PROGRAM LateBlanking_Scan
VAR
	CS_CodeTcp_cold: CS_CodeTcp;
	Cold_step :UINT;
	scan_TON1 :Tc2_Standard.TON;
	Scan_TON :ARRAY[1..7] OF Tc2_Standard.TON;
	Scan_code_Z : R_TRIG;
	I:INT;
END_VAR

//扫码



Saoma();
P3User2_Par.Scan_IP:='192.168.10.26';
Scan_TON[1](PT:=T#1MS);
Scan_TON[2](PT:=T#1MS);
Scan_TON[3](PT:=T#1MS);
Scan_TON[4](PT:=T#100MS);

Scan_code_Z (CLK:=Cold_Scan_code, Q=>);

IF Scan_code_Z.Q AND  Cold_step=0 THEN
	 Cold_step:=10;
END_IF




CASE Cold_step OF
0:
	IF Scan_start AND NOT bCodeError AND NOT bCodeConError AND NOT P3User2_Par.Shield[4] THEN
	 Cold_step:=10;
	 Code_State:=0;
	ELSIF P3User2_Par.Shield[4] THEN
	 Cold_step:=70;
	END_IF
10:
	Scan_TON[1].IN:=FALSE;
	Scan_TON[2].IN:=FALSE;
	Scan_TON[3].IN:=FALSE;
	Cold_step:=20;
	
20:
	bScan_init:=TRUE;
	Scan_TON[1].IN:=TRUE;
	IF Scan_TON[1].Q THEN
		bScan_init:=FALSE;
		Scan_TON[1].IN:=FALSE;
		Cold_step:=30;
	END_IF

30:
	bTcpOpen:=TRUE;
	Scan_TON[2].IN:=TRUE;
	IF Scan_TON[2].Q THEN
		bTcpOpen:=FALSE;
		Scan_TON[2].IN:=FALSE;
		Cold_step:=40;
	END_IF

40:
	IF bTcpOpen_OK THEN
		Cold_step:=50;
	END_IF

50:
	bScan_start:=TRUE;
	Scan_TON[3].IN:=TRUE;
	IF Scan_TON[3].Q THEN
		bScan_start:=FALSE;
		Scan_TON[3].IN:=FALSE;
		Cold_step:=60;
	END_IF
60:
	Scan_TON[4].IN:=TRUE;
	IF 	Scan_TON[4].Q THEN
		Cold_step:=70;
		Scan_TON[4].IN:=FALSE;
	END_IF

70:
IF NOT P3User2_Par.Shield[4] THEN
	IF Code_State=1 AND (strCode<>'') THEN
		CellMemory[CellNo.OvenMoveClip1].Cell_number1:=strCode;
		IF strCode=CellMemory[CellNo.OvenMoveClip1].Cell_number THEN
			CellMemory[CellNo.OvenMoveClip1].ScanCode:=1;
			Scan_start:=FALSE;
			Scan_finish:=TRUE;
			Cold_step:=80;				
			I:=0;
		ELSIF strCode<>CellMemory[CellNo.OvenMoveClip1].Cell_number THEN
			CellMemory[CellNo.OvenMoveClip1].ScanCode:=2;
			P3_Error[79]:=TRUE;//冷压扫码第二次扫码校验NG
			Scan_start:=FALSE;
			Scan_finish:=TRUE;
			Cold_step:=80;
			I:=0;
		END_IF
	ELSIF  Code_State=2 AND I<3 THEN
			Cold_step:=10;
			I:=I+1;		
	ELSIF Code_State=2 AND I>=3 THEN
		CellMemory[CellNo.ColdpressClip].Cell_number1:=strCode;
		CellMemory[CellNo.ColdpressClip].ScanCode:=2;
		P3_Error[16]:=TRUE;//冷压扫码NG报警
		Scan_start:=FALSE;
		Scan_finish:=TRUE;
		Cold_step:=80;
		I:=0;
	END_IF
ELSIF P3User2_Par.Shield[4] THEN
		CellMemory[CellNo.OvenMoveClip1].Cell_number1:='A1234567890ABCDEF';
		CellMemory[CellNo.OvenMoveClip1].ScanCode:=1;
		Scan_start:=FALSE;
		Scan_finish:=TRUE;
		Cold_step:=80;				
		I:=0;
END_IF
80:
	IF NOT Scan_finish THEN
		Cold_step:=0;
	END_IF
END_CASE

ACTION Saoma:
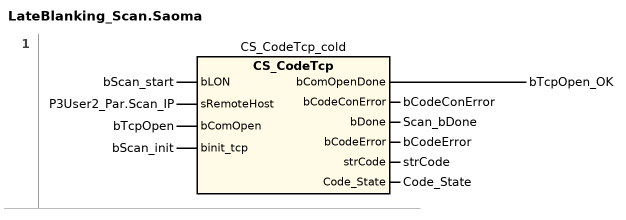
// NETWORK 1
CS_CodeTcp_cold(
    bLON := bScan_start,
    sRemoteHost := P3User2_Par.Scan_IP,
    bComOpen := bTcpOpen,
    binit_tcp := bScan_init,
    bCodeConError => bCodeConError,
    bDone => Scan_bDone,
    bCodeError => bCodeError,
    strCode => strCode,
    Code_State => Code_State); // CS_CodeTcp
bTcpOpen_OK := CS_CodeTcp_cold.bComOpenDone;
END_ACTION

END_PROGRAM

(* stored: Version 1.1.0.1, ProductVersion 3.1.4024.12
   POU LateBlanking_Scan: Id {ce93b600-106b-40b8-920f-d09054d889b5}, SpecialFunc None
   Action Saoma: Id {45f5bdef-7600-46ac-a803-74a1b2ec8b7c} *)
